TYPE FILE_ACTION :
STRUCT
	Id : UINT;
END_STRUCT
END_TYPE

(* stored: Version 1.1.0.1
   DUT FILE_ACTION: Id {b66da3d6-15de-438d-870d-8307bde7b67a} *)
